FUNCTION_BLOCK TrackingLogic
VAR_INPUT
END_VAR
VAR_OUTPUT
END_VAR
VAR
	target_ID : INT;
END_VAR

target_ID := AUTO.Stages[AUTO.Recept][AUTO.StageSelect].I;
IF target_ID <> 0 AND AUTO.Current.P > 13 THEN
	AUTO.VRoki := target_ID;
	GVL.LEDLBlue := TRUE;
END_IF
IF AUTO.Current.P < 5 THEN
	AUTO.VRoki := 0;
	GVL.LEDLBlue := 0;
END_IF

IF AUTO.VRoki <> 0 THEN
	AUTO.Items[AUTO.VRoki].A := AUTO.Current.A;
	AUTO.Items[AUTO.VRoki].Y := AUTO.Current.Y;
	AUTO.Items[AUTO.VRoki].Z := AUTO.Current.Z; 
END_IF

END_FUNCTION_BLOCK

(* stored: Version 1.1.0.1, ProductVersion 3.1.4024.12
   POU TrackingLogic: Id {08bd7de2-ed34-413b-853a-e57239f0a725}, SpecialFunc None *)
